PROGRAM MAIN
VAR
	I0_0 : BOOL;
    Q0_0 : BOOL;
END_VAR

END_PROGRAM

(* stored: Version 1.1.0.1, ProductVersion 3.1.4024.16
   POU MAIN: Id {cd1d376f-9eac-485c-84d7-1fbf9a64bde5}, SpecialFunc None *)
